VAR_GLOBAL CONSTANT
	iMAX_AXES_REF : INT := 5;
END_VAR

VAR_GLOBAL
	iGlobalCounter : UINT;
	fbCrititcalSection : FB_IecCriticalSection;
END_VAR

VAR_GLOBAL
	{attribute 'TcContextName':='NC SAF'}
	Nc2MasterAxis : Tc2_MC2.AXIS_REF;
END_VAR

(* stored: Version 1.1.0.1
   GVL GVL: Id {b31223e4-d801-463b-aea4-2814692ede38} *)
